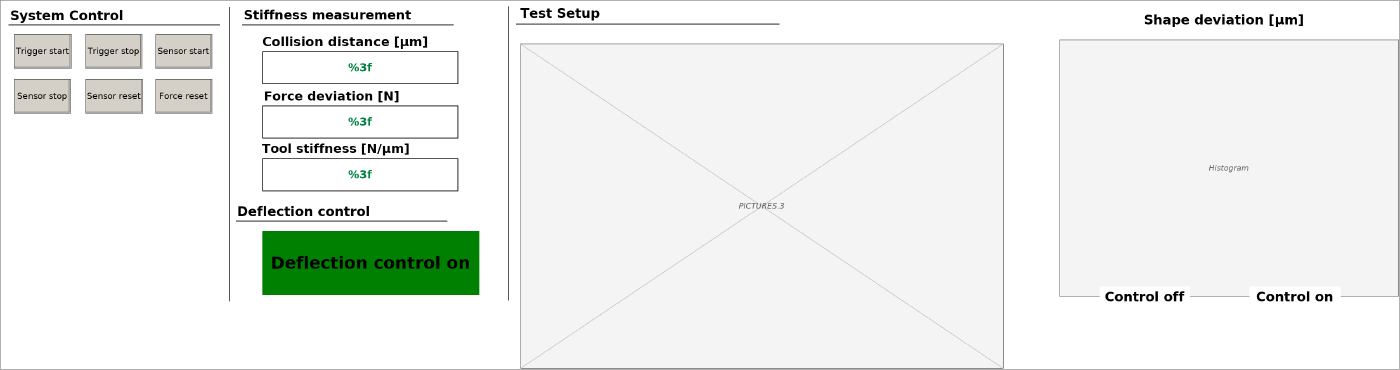
VISUALIZATION VISUALISATION_EMO2017  // 1804x477
    Rectangle (338,298 279x82), "Deflection control off", invisible if: 1
    Button (18,44 74x44), "Trigger start"
        OnMouseClick: execute { VARIABLES.CAN_TRIGGER_STATE:=1; }
    Button (110,44 73x44), "Trigger stop"
        OnMouseClick: execute { VARIABLES.CAN_TRIGGER_STATE:=0; }
    Button (200,44 73x44), "Sensor start"
        OnMouseClick: execute { CAN_CONTROL_STATE:=1; }
    Button (18,102 73x44), "Sensor stop"
        OnMouseClick: execute { CAN_CONTROL_STATE:=0; }
    Button (110,102 74x44), "Sensor reset"
        OnMouseClick: execute { CAN_CONTROL_STATE:=2; }
    Button (200,102 73x44), "Force reset"
        OnMouseClick: execute { FORCE_RESET:=1; }
    Rectangle (11,5 150x30), "System Control"
    Rectangle (313,12 218x15), "Stiffness measurement"
    Rectangle (338,204 252x42), "%3f", text variable: VARIABLES.TOOL_STIFFNESS[1]
    Rectangle (338,66 252x42), "%3f", text variable: VARIABLES.COLLISION_DISTANCE
    Rectangle (338,136 252x42), "%3f", text variable: VARIABLES.FORCE_DEVIATION[1]
    Rectangle (337,44 216x20), "Collision distance [µm]"
    Rectangle (340,114 175x20), "Force deviation [N]"
    Rectangle (338,183 190x17), "Tool stiffness [N/µm]"
    Line (295,9) (295,388)
    Line (584,32) (312,32)
    Group (1365,12 437x384)
        Histogram (0,39 437x331), scale format: %.1f, scale 0..50
            p1518820177: VARIABLES.RESULT
            p102497268: VARIABLES.RESULT
            p788070771: ARRAY [1..2] OF REAL
        Rectangle (245,357 117x27), "Control on"
        Rectangle (52,357 116x27), "Control off"
        Rectangle (110,0 205x27), "Shape deviation [µm]"
    Line (283,32) (11,32)
    Image (670,56 623x419), image: PICTURES.3
    Rectangle (654,-2 136x38), "Test Setup"
    Line (1004,31) (665,31)
    Line (655,8) (655,387)
    Line (576,285) (304,285)
    Rectangle (301,265 181x15), "Deflection control"
    Rectangle (338,298 279x82), "Deflection control on", invisible if: DEFLECTION_CONTROL_ON<>1
END_VISUALIZATION

(* stored: Version 1.1.0.1, ProductVersion 3.1.4022.16
   Visu VISUALISATION_EMO2017: Id {7b254422-13a8-400e-a5a3-2b488a96be65} *)
